TYPE g_ttrrr:
    STRUCT
        field1: g_trr;
        field2: REAL;
    END_STRUCT;
END_TYPE
